// TIA Portal V18 export
TYPE "UDT_Stopper_FB"
// stored: IsFailsafeCompliant false
   STRUCT
      In : Struct
         iSensor : Bool;   // 本站托盘到位
         iNextSensor : Bool;   // 后站托盘到位
         iNextValve : Bool;   // 后站挡停输出
         iPresentDwell : Time := T#0.3s;   // 本站到位传感器延时
         iNextEmptyDwell : Time := T#10s;   // 后站托盘到位传感器延时
         iReleaseClear : Bool;   // 托盘释放允许
         iReleaseDwell : Time := T#1s;   // 托盘已流出延时
         iReleaseFaultTimer : Time := T#1s;   // 托盘流出超时延时
         iReachFaultTimer : Time := T#5s;   // 托盘流入后站超时延时
      END_STRUCT;
      Out : Struct
         oValve : Bool;   // 本站挡停输出
         oReleaseCompleted : Bool;   // 释放完成
         oReleaseFault : Bool;   // 托盘流走超时
         oReachFault : Bool;   // 后站托盘接收超时
         oNotClear : Bool;   // 手动释放中
      END_STRUCT;
   END_STRUCT;
END_TYPE
